// TIA Portal V16 export
// export: Created 2021-04-06T19:52:16.7316094Z, ExportSetting WithDefaults, DisplayName Totally Integrated Automation Portal, DisplayVersion V16, DisplayName TIA Portal Version Control Interface, DisplayVersion V16, DisplayName TIA Portal Openness, DisplayVersion V16, DisplayName STEP 7 Professional, DisplayVersion V16, DisplayName STEP 7 Safety, DisplayVersion V16, DisplayName WinCC Unified SCADA Engineering System, DisplayVersion V16
FUNCTION_BLOCK "workPackingMachine_AM"   // FB4, LAD
TITLE = Работа с УМ, бункерами
{ S7_Optimized_Access := 'TRUE' }
VERSION : 0.1
// stored: AutoNumber true, IsIECCheckEnabled false, IsRetainMemResEnabled false, MemoryReserve 100, SetENOAutomatically false, UDAEnableTagReadback false
   VAR_INPUT
      enWork : Bool;   // разрешение работы
      YP_ReadyAccept : Array[0..2] of Bool;   // сигнал от упак машины что готова принять
      YP_StartDozing : Array[0..2] of Bool;   // сигнал от упаковочной машины что начать дозирование
      weightPack : Real;   // заданный вес упаковки
   END_VAR
   VAR_IN_OUT
      hmiYpDropWeight : Array[0..2] of Real;   // вывод на панель сброшенного веса
      hmiYPDropErrorMeasure : Array[0..2] of Real;   // вывод на панель погрешности
      openLeftBunker : Array[0..12] of Bool;   // сгналы открытия левых бункеров
      closeLeftBunker : Array[0..12] of Bool;   // сигналы закрытия левых бункеров
      openRightBunker : Array[0..12] of Bool;   // сигналы открытия правых бункеров
      closeRightBunker : Array[0..12] of Bool;   // сигналы закрытия правых бункеров
      alarmStop : Bool;   // аварийный останов
      Yq_ReadyDoze : Array[0..2] of Bool;   // сигнал на упаковочную машину что доза готова
      YP_ReadyToDrop : Array[0..2] of Bool;   // сигнал говорит о том что в УМ можно 100% чтото скинуть
      stableWeightBunker : Array[0..12] of Real;   // стабильный вес в бункерах
      readyToSort : Array[0..12] of Bool;
      readyToDrop : Array[0..12] of Bool;   // массив который будет сбрасываться
      Conv_FRV : Array[0..2] of Bool;   // запуск конвейеров вперед
      Conv_REV : Array[0..2] of Bool;   // запуск конвейеров назад
   END_VAR
   VAR
      dropLeftBunker { ExternalAccessible := 'False'; ExternalVisible := 'False'; ExternalWritable := 'False'} : Array[0..12] of Bool;   // массив на сброс левых бункеров
      dropRightBunker { ExternalAccessible := 'False'; ExternalVisible := 'False'; ExternalWritable := 'False'} : Array[0..12] of Bool;   // массив на сброс правых бункеров
      tmpPtrig : Array[0..1] of Bool;
      dropTon : Array[0..2] of TON_TIME;   // выдержка на передачу сигнала УМ ДОЗА
      startDropTon : Array[0..2] of Bool;   // начало отсчета для таймера
      dropWeight : Real;   // сбрасываемый вес
      nextDropConveyer : SInt;   // индекс конвейера на который сбрасывали последним
      tonReadyDozeTimer : Array[0..2] of TON_TIME;
      leftBunker_FB : Array[0..12] of "controlValve";
      rightBunker_FB : Array[0..12] of "controlValve";
      full1 : Array[0..12] of Bool;
      full0 : Array[0..12] of Bool;
      valueDropBunker : Bool;
      watchDrop : Array[0..12] of Bool;
   END_VAR
   VAR_TEMP
      i : SInt;
      resetTimerDropYp : Array[0..2] of Bool;
      resetTimerDropTon : Array[0..2] of Bool;
   END_VAR
   // full1[1..12] := true;
   VAR_TEMP   // added for the SCL form of the ladder/FBD networks
      _w1 : Bool;
      _w2 : Bool;
   END_VAR
BEGIN

REGION Network 1: сброс вращения если убрать сигнал разрешения
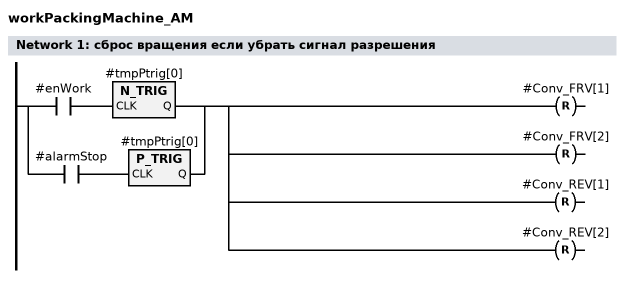
   RUNG wire#powerrail
      Contact( #enWork )
      N_Trig( #tmpPtrig[0] )
      wire#w1
      R_Coil( #Conv_FRV[1] )
   END_RUNG
   RUNG wire#powerrail
      Contact( #alarmStop )
      P_Trig( #tmpPtrig[0] )
   END_RUNG wire#w1
   RUNG wire#w1
      R_Coil( #Conv_FRV[2] )
   END_RUNG
   RUNG wire#w1
      R_Coil( #Conv_REV[1] )
   END_RUNG
   RUNG wire#w1
      R_Coil( #Conv_REV[2] )
   END_RUNG
   // the same network as SCL:
   #_w1 := NOT #enWork AND #tmpPtrig[0];   // falling edge
   #tmpPtrig[0] := #enWork;
   #_w2 := #alarmStop AND NOT #tmpPtrig[0];   // rising edge
   #tmpPtrig[0] := #alarmStop;
   IF #_w1 OR #_w2 THEN
       #Conv_FRV[1] := FALSE;
       #Conv_FRV[2] := FALSE;
       #Conv_REV[1] := FALSE;
       #Conv_REV[2] := FALSE;
   END_IF;
END_REGION

REGION Network 2 (SCL): Подсчет сбрасываемых бункеров
   #i := 0;
   #valueDropBunker := FALSE;
   FOR #i := 1 TO 12 DO
       IF #readyToDrop[#i] THEN
           #valueDropBunker := true;
           EXIT;
       END_IF;
   END_FOR;
END_REGION

REGION Network 3 (SCL): Сброс сигнала на УМ #Yq_ReadyDoze
   #i := 0;
   FOR #i := 1 TO 2 DO
       // IF #Yq_ReadyDoze[#i] THEN
       //     #Yq_ReadyDoze[#i] := false;
       // END_IF;
       #tonReadyDozeTimer[#i](IN := #Yq_ReadyDoze[#i],
                              PT := t#1s,
                              Q=>#resetTimerDropYp[#i]);

   END_FOR;
   #i := 0;
   FOR #i := 1 TO 2 DO

       IF #resetTimerDropYp[#i] THEN
           #Yq_ReadyDoze[#i] := false;
       END_IF;

   END_FOR;
END_REGION

REGION Network 4 (SCL): Формирование сигналов
   // #YP_ReadyToDrop
   #i := 0;
   FOR #i := 1 TO 2 DO
       #YP_ReadyToDrop[#i] := #YP_ReadyAccept[#i] AND #YP_StartDozing[#i] AND NOT(#startDropTon[#i]) AND NOT(#Yq_ReadyDoze[#i]);
   END_FOR;
END_REGION

REGION Network 5 (SCL): учет сбрасываемого веса
   // помещаем в переменнную #dropWeight вес который будет сброшен
   IF #enWork THEN
       IF (#YP_ReadyToDrop[1] OR #YP_ReadyToDrop[2]) AND #valueDropBunker  THEN
           #i := 0;
           FOR #i := 1 TO 12 DO
               #dropWeight := #dropWeight + BOOL_TO_INT(#readyToDrop[#i])
               * #stableWeightBunker[#i];
           END_FOR;
       END_IF;
   END_IF;
END_REGION

REGION Network 6 (SCL): вращение конвейеров
   //"hmi".outConvAndPack[1].isUseInBegin - разрешение использовать
   // "hmi".outConvAndPack[1].isUpInBegin - вращать вперед
   #i := 0;
   FOR #i := 1 TO 2 DO
       IF #enWork AND "hmi".outConvAndPack[#i].isUseInBegin THEN
           IF "hmi".outConvAndPack[#i].isUpInBegin THEN
               #Conv_FRV[#i] := true;
               #Conv_REV[#i] := false;
           ELSE
               #Conv_FRV[#i] := false;
               #Conv_REV[#i] := true;
           END_IF;
       ELSE
           #Conv_FRV[#i] := false;
           #Conv_REV[#i] := false;
       END_IF;
   END_FOR;
END_REGION

REGION Network 7 (SCL): Формирование сигнала доза готова
   IF #enWork THEN
       IF #valueDropBunker THEN//определяем какие бункеры открываем
           //, а также даем отсечку времени для отправки
           //ДОЗА ГОТОВА
           IF #YP_ReadyToDrop[1] OR #YP_ReadyToDrop[2] THEN
               //ПРОСТО ЕСЛИ НЕ СКИДЫВАЕМ ТО И НЕ НАДО ОЧИЩАТЬ МАССИВ READYTOdROP
               IF #YP_ReadyToDrop[1] AND #YP_ReadyToDrop[2] THEN
                   //если оба доступны то по следующему индексу
                   CASE #nextDropConveyer OF
                       0, 2:  //следующий был второй
                           IF #Conv_FRV[2] THEN
                               #hmiYpDropWeight[1] := #dropWeight;
                               #hmiYPDropErrorMeasure[1] := (#weightPack - #dropWeight) / #weightPack * 100;
                               #startDropTon[1] := true;
                           ELSE
                               #hmiYpDropWeight[2] := #dropWeight;
                               #hmiYPDropErrorMeasure[2] := (#weightPack - #dropWeight) / #weightPack * 100;
                               #startDropTon[2] := true;
                           END_IF;
                           #dropLeftBunker := #readyToDrop;

                       1:  // следующий первый
                           IF #Conv_FRV[1] THEN
                               #hmiYpDropWeight[1] := #dropWeight;
                               #hmiYPDropErrorMeasure[1] := (#weightPack - #dropWeight) / #weightPack * 100;
                               #startDropTon[1] := true;
                           ELSE
                               #hmiYpDropWeight[2] := #dropWeight;
                               #hmiYPDropErrorMeasure[2] := (#weightPack - #dropWeight) / #weightPack * 100;
                               #startDropTon[2] := true;
                           END_IF;
                           #dropRightBunker := #readyToDrop;

                   END_CASE;

               ELSE
                   #i := 0;
                   FOR #i := 1 TO 2 DO
                       IF #YP_ReadyToDrop[#i] THEN
                           #hmiYpDropWeight[#i] := #dropWeight;
                           #hmiYPDropErrorMeasure[#i] := (#weightPack - #dropWeight) / #weightPack * 100;
                           #startDropTon[#i] := TRUE;

                           IF (#Conv_FRV[1] AND #Conv_FRV[2]) OR //если конвейера вращаются в одну сторону
                               (#Conv_REV[1] AND #Conv_REV[2]) THEN
                               #dropLeftBunker := #readyToDrop;
                               #dropRightBunker := #readyToDrop;
                               #watchDrop := #readyToDrop;
                           ELSE
                               IF #i = 1 THEN//Если готова только первая УМ
                                   IF #Conv_FRV[1] THEN
                                       #dropRightBunker := #readyToDrop;
                                   ELSE
                                       #dropLeftBunker := #readyToDrop;
                                   END_IF;
                               ELSE//если готова только вторая УМ
                                   IF #Conv_REV[1] THEN
                                       #dropRightBunker := #readyToDrop;
                                   ELSE
                                       #dropLeftBunker := #readyToDrop;
                                   END_IF;

                               END_IF;

                           END_IF;
                           EXIT;//выйти из for если нашли нужную УМ
                       END_IF;
                   END_FOR;
               END_IF;
               #readyToDrop := #full0;
           END_IF;
       END_IF;
   END_IF;

   //изменяем конвейер на который будем скидывать
   IF #dropWeight >= #weightPack AND (#YP_ReadyToDrop[1] OR #YP_ReadyToDrop[2])THEN
       #dropWeight := 0;
       IF #nextDropConveyer = 0 OR #nextDropConveyer = 2 THEN
           #nextDropConveyer := 1;
       ELSE
           #nextDropConveyer := 2;
       END_IF;
   END_IF;
END_REGION

REGION Network 8 (SCL): открывание левых и правых бункеров
   IF #enWork THEN
       #i := 0;
       FOR #i := 1 TO 12 DO

           #leftBunker_FB[#i](autoclose_M := TRUE,
                             time_autoclose := T#500ms,
                             "time_open/close" := T#200ms,
                             openQ => #openLeftBunker[#i],
                             closeQ => #closeLeftBunker[#i],
                             open := #dropLeftBunker[#i],
                             stopAlarm := #alarmStop);
           #dropLeftBunker[#i] := false;


           #rightBunker_FB[#i](autoclose_M := TRUE,
                              time_autoclose := T#500ms,
                              "time_open/close" := T#200ms,
                              openQ => #openRightBunker[#i],
                              closeQ => #closeRightBunker[#i],
                              open := #dropRightBunker[#i],
                              stopAlarm := #alarmStop);
           #dropRightBunker[#i] := false;

       END_FOR;
   END_IF;
END_REGION

REGION Network 9 (SCL): Формирование сигнала ДОЗА на упаковочную машину
   #i := 0;
   FOR #i := 1 TO 2 DO
       #dropTon[#i](IN := #startDropTon[#i],
                    PT := t#1500ms,
                    Q=>#resetTimerDropTon[#i]);

       IF #resetTimerDropTon[#i] THEN
           #Yq_ReadyDoze[#i] := true;
           #startDropTon[#i] := false;
       END_IF;

       "hmi".outConvAndPack[#i].isReadyDozaPackingMachine := #Yq_ReadyDoze[#i];
   END_FOR;
END_REGION
END_FUNCTION_BLOCK
